TEXTLIST TXT_LIST_OP_MODE
  7 = 'NOT-HALT' | en: 'EMERGANCY-STOP' | de: 'NOT-HALT' | zh_CHS: '急停'
  8 = 'MASCHINEN-FEHLER' | en: 'FATAL ERROR' | de: 'MASCHINEN-FEHLER' | zh_CHS: '致命错误'
  9 = 'STEUERUNG EIN' | en: 'CONTROL ON' | de: 'STEUERUNG EIN' | zh_CHS: '控制开启'
  1 = 'AUTOMATIK ' | en: 'AUTOMATIC' | de: 'AUTOMATIK ' | zh_CHS: '自动'
  2 = 'HANDBETRIEB' | en: 'MANUAL MODE' | de: 'HANDBETRIEB' | zh_CHS: '手动模式'
  3 = 'TIPPBETRIEB' | en: 'DEBUG MODE' | de: 'TIPPBETRIEB' | zh_CHS: 'DEBUG MODE'
  4 = 'GRUNDSTELLUNGSFAHRT' | en: 'INITIAL POS RIDE' | de: 'GRUNDSTELLUNGSFAHRT' | zh_CHS: '复位'
  5 = 'GRUNDSTELLUNG ERREICHT' | en: 'INITIAL POS REACH' | de: 'GRUNDSTELLUNG ERREICHT' | zh_CHS: '达成基本要求'
  101 = 'GST' | en: 'INIT' | de: 'GST' | zh_CHS: '的INIT'
  102 = 'AUTO' | en: 'AUTO' | de: 'AUTO' | zh_CHS: '自动'
  103 = 'HAND' | en: 'MANUAL' | de: 'HAND' | zh_CHS: '手册'
  104 = 'TIPP' | en: 'DEBUG' | de: 'TIPP' | zh_CHS: '去调查'
  105 = 'START' | en: 'START' | de: 'START' | zh_CHS: '开始'
  106 = 'STOP' | en: 'STOP' | de: 'STOP' | zh_CHS: '停'
  11 = 'VORWAHL AUTOMATIK' | en: 'SELECTION AUTOMATIC' | de: 'VORWAHL AUTOMATIK' | zh_CHS: '自动选择'
  12 = 'VORWAHL HAND' | en: 'SELECTION MANUAL' | de: 'VORWAHL HAND' | zh_CHS: '选择手册'
  13 = 'VORWAHL TIPPBETRIEB' | en: 'SELECTION DEBUG' | de: 'VORWAHL TIPPBETRIEB' | zh_CHS: '选择调试'
  14 = 'VORWAHL GRUNDSTELLUNGSFAHRT' | en: 'SLECTION INITIAL POS RIDE' | de: 'VORWAHL GRUNDSTELLUNGSFAHRT' | zh_CHS: '选择初始POS RIDE'
  0 = 'MASCHINE EINSCHALTEN' | en: 'TURN ON THE MACHINE' | de: 'MASCHINE EINSCHALTEN' | zh_CHS: '启动机器'
  107 = 'PAUSE' | en: 'PAUSE' | de: 'PAUSE'
  6 = 'PAUSE' | en: 'PAUSE' | de: 'PAUSE'
  10 = 'DRUCK OK' | en: 'DRUCK OK' | de: 'MAIN AIR OK'
   = ''
END_TEXTLIST

(* stored: Version 1.1.0.1, ProductVersion 3.1.4024.12
   TextList TXT_LIST_OP_MODE: Id {d99f2127-786d-40dc-b5f2-fb061556cfe7} *)
